TYPE ST_EL6910 :
STRUCT
	
	// TERMINAL - EL6910	TwinSAFE logic	 (Term 3)
	sTerminalName                                           :   STRING(200):= 'EL6910 | TwinSAFE logic';
	stTerminalInfo											: 	ST_Terminal_Info;

END_STRUCT
END_TYPE

(* stored: Version 1.1.0.1, ProductVersion 3.1.4024.13
   DUT ST_EL6910: Id {88323c5e-5169-4252-81dd-45e9b175c575} *)
